TYPE
  (* Standard: 61499-1 *)
  (* Version 1.0, 2026-06-15, Dimitrios Kalligaridis *)
  PACKAGE mypackage;
  MyStruct : STRUCT
    A : BOOL;
    B : BOOL;
  END_STRUCT;
END_TYPE
